FUNCTION_BLOCK Relay
VAR
	bOutput	AT%Q*	: BOOL;
	tonPulse		: TON;
END_VAR

METHOD Pulse : BOOL
VAR_INPUT
	tPulseTime	: TIME;
END_VAR
tonPulse(IN := TRUE, PT:= tPulseTime);

IF NOT tonPulse.Q THEN
	SwitchOn();
ELSIF tonPulse.Q THEN
	SwitchOff();
	tonPulse(IN := FALSE);
	Pulse := TRUE;
END_IF
END_METHOD

METHOD SwitchOff : BOOL
VAR_INPUT
END_VAR
bOutput := FALSE;

SwitchOff := TRUE;
END_METHOD

METHOD SwitchOn : BOOL
VAR_INPUT
END_VAR
bOutput := TRUE;

SwitchOn := TRUE;
END_METHOD

END_FUNCTION_BLOCK

(* stored: Version 1.1.0.1
   POU Relay: Id {5085b1cf-4d06-4906-8007-1329dfffaf0f}, SpecialFunc None
   Method Pulse: Id {1937db57-4c05-4d40-92ff-67b59d714bee}
   Method SwitchOff: Id {71d54ee8-6e93-447d-8209-bf17b3119904}
   Method SwitchOn: Id {c87da857-2505-48e7-b65d-b923003a41ae} *)
